// TIA Portal V19 export
FUNCTION "INTERLOCK" : Void   // FC7, LAD
{ S7_Optimized_Access := 'TRUE' }
// stored: SetENOAutomatically false
   VAR_TEMP   // added for the SCL form of the ladder/FBD networks
      _w1 : Bool;
      _w2 : Bool;
   END_VAR
BEGIN

REGION Network 1: ERROR
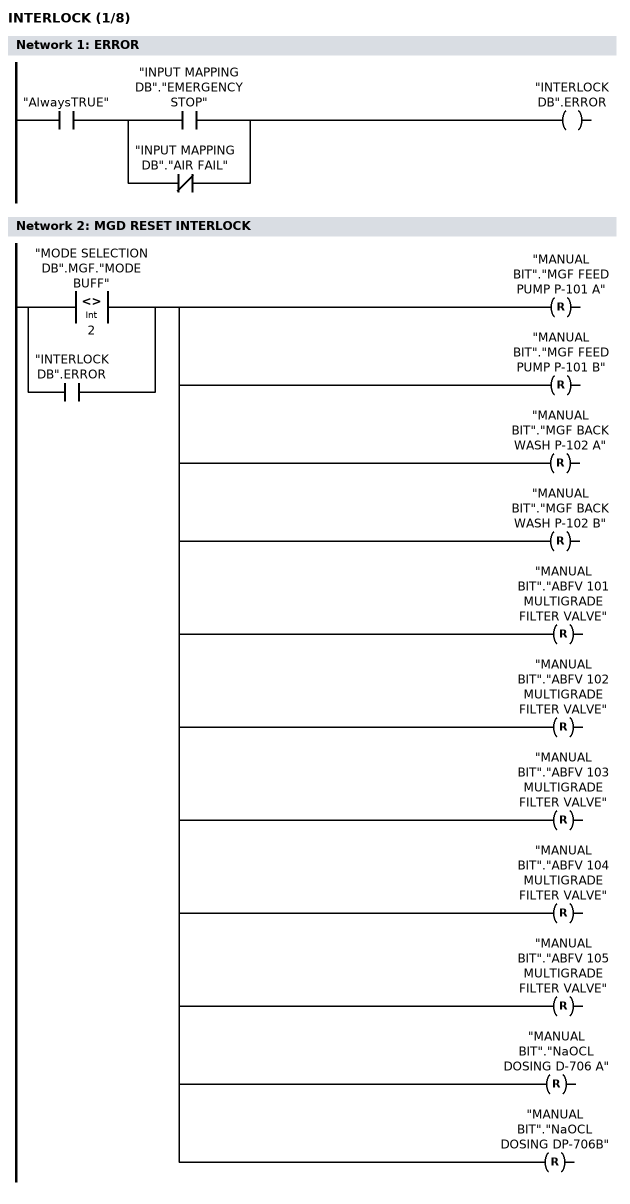
   RUNG wire#powerrail
      Contact( "AlwaysTRUE" )
      wire#w1
      Contact( "INPUT MAPPING DB"."EMERGENCY STOP" )
      wire#w2
      Coil( "INTERLOCK DB".ERROR )
   END_RUNG
   RUNG wire#w1
      I_Contact( "INPUT MAPPING DB"."AIR FAIL" )
   END_RUNG wire#w2
   // the same network as SCL:
   "INTERLOCK DB".ERROR := "AlwaysTRUE" AND ("INPUT MAPPING DB"."EMERGENCY STOP" OR NOT "INPUT MAPPING DB"."AIR FAIL");
END_REGION

REGION Network 2: MGD RESET INTERLOCK
   RUNG wire#powerrail
      { S7_Templates := "SrcType := Int" } NE_Contact(in1 := "MODE SELECTION DB".MGF."MODE BUFF", in2 := 2)
      wire#w1
      R_Coil( "MANUAL BIT"."MGF FEED PUMP P-101 A" )
   END_RUNG
   RUNG wire#powerrail
      Contact( "INTERLOCK DB".ERROR )
   END_RUNG wire#w1
   RUNG wire#w1
      R_Coil( "MANUAL BIT"."MGF FEED PUMP P-101 B" )
   END_RUNG
   RUNG wire#w1
      R_Coil( "MANUAL BIT"."MGF BACK WASH P-102 A" )
   END_RUNG
   RUNG wire#w1
      R_Coil( "MANUAL BIT"."MGF BACK WASH P-102 B" )
   END_RUNG
   RUNG wire#w1
      R_Coil( "MANUAL BIT"."ABFV 101 MULTIGRADE FILTER VALVE" )
   END_RUNG
   RUNG wire#w1
      R_Coil( "MANUAL BIT"."ABFV 102 MULTIGRADE FILTER VALVE" )
   END_RUNG
   RUNG wire#w1
      R_Coil( "MANUAL BIT"."ABFV 103 MULTIGRADE FILTER VALVE" )
   END_RUNG
   RUNG wire#w1
      R_Coil( "MANUAL BIT"."ABFV 104 MULTIGRADE FILTER VALVE" )
   END_RUNG
   RUNG wire#w1
      R_Coil( "MANUAL BIT"."ABFV 105 MULTIGRADE FILTER VALVE" )
   END_RUNG
   RUNG wire#w1
      R_Coil( "MANUAL BIT"."NaOCL DOSING D-706 A" )
   END_RUNG
   RUNG wire#w1
      R_Coil( "MANUAL BIT"."NaOCL DOSING DP-706B" )
   END_RUNG
   // the same network as SCL:
   IF ("MODE SELECTION DB".MGF."MODE BUFF" <> 2) OR "INTERLOCK DB".ERROR THEN
       "MANUAL BIT"."MGF FEED PUMP P-101 A" := FALSE;
       "MANUAL BIT"."MGF FEED PUMP P-101 B" := FALSE;
       "MANUAL BIT"."MGF BACK WASH P-102 A" := FALSE;
       "MANUAL BIT"."MGF BACK WASH P-102 B" := FALSE;
       "MANUAL BIT"."ABFV 101 MULTIGRADE FILTER VALVE" := FALSE;
       "MANUAL BIT"."ABFV 102 MULTIGRADE FILTER VALVE" := FALSE;
       "MANUAL BIT"."ABFV 103 MULTIGRADE FILTER VALVE" := FALSE;
       "MANUAL BIT"."ABFV 104 MULTIGRADE FILTER VALVE" := FALSE;
       "MANUAL BIT"."ABFV 105 MULTIGRADE FILTER VALVE" := FALSE;
       "MANUAL BIT"."NaOCL DOSING D-706 A" := FALSE;
       "MANUAL BIT"."NaOCL DOSING DP-706B" := FALSE;
   END_IF;
END_REGION

REGION Network 3: UF RESET INTERLOCK
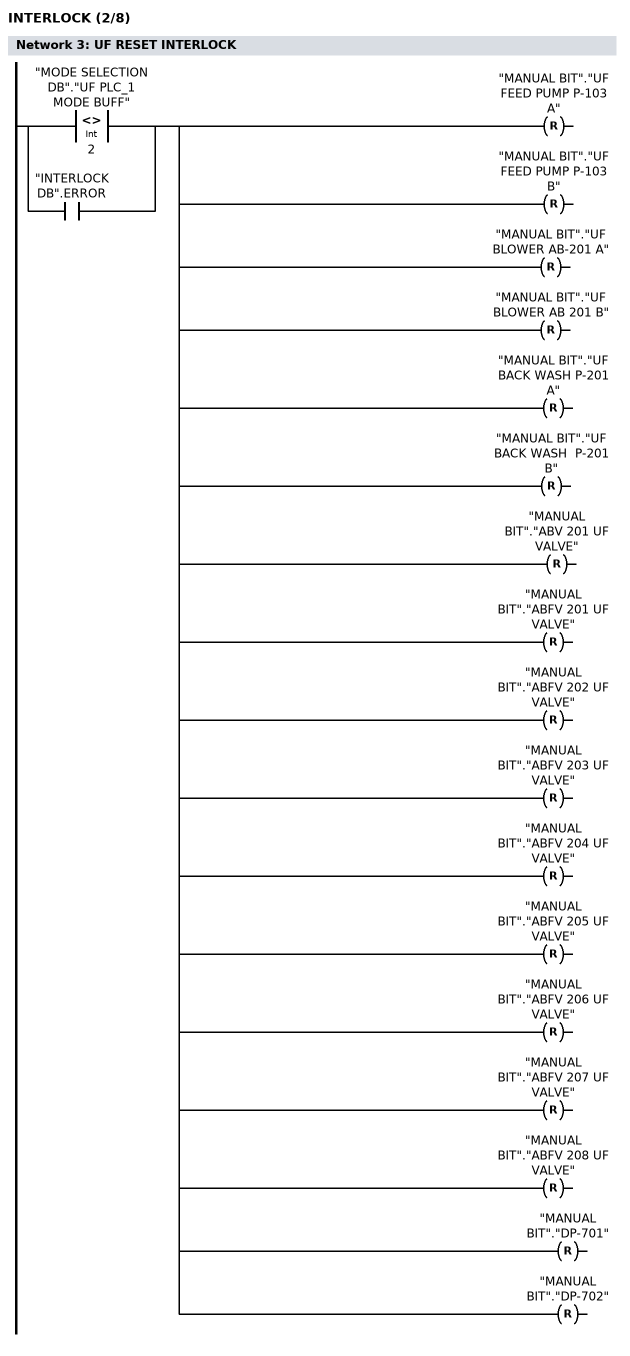
   RUNG wire#powerrail
      { S7_Templates := "SrcType := Int" } NE_Contact(in1 := "MODE SELECTION DB"."UF PLC_1 MODE BUFF", in2 := 2)
      wire#w1
      R_Coil( "MANUAL BIT"."UF FEED PUMP P-103 A" )
   END_RUNG
   RUNG wire#powerrail
      Contact( "INTERLOCK DB".ERROR )
   END_RUNG wire#w1
   RUNG wire#w1
      R_Coil( "MANUAL BIT"."UF FEED PUMP P-103 B" )
   END_RUNG
   RUNG wire#w1
      R_Coil( "MANUAL BIT"."UF BLOWER AB-201 A" )
   END_RUNG
   RUNG wire#w1
      R_Coil( "MANUAL BIT"."UF BLOWER AB 201 B" )
   END_RUNG
   RUNG wire#w1
      R_Coil( "MANUAL BIT"."UF BACK WASH P-201 A" )
   END_RUNG
   RUNG wire#w1
      R_Coil( "MANUAL BIT"."UF BACK WASH  P-201 B" )
   END_RUNG
   RUNG wire#w1
      R_Coil( "MANUAL BIT"."ABV 201 UF VALVE" )
   END_RUNG
   RUNG wire#w1
      R_Coil( "MANUAL BIT"."ABFV 201 UF VALVE" )
   END_RUNG
   RUNG wire#w1
      R_Coil( "MANUAL BIT"."ABFV 202 UF VALVE" )
   END_RUNG
   RUNG wire#w1
      R_Coil( "MANUAL BIT"."ABFV 203 UF VALVE" )
   END_RUNG
   RUNG wire#w1
      R_Coil( "MANUAL BIT"."ABFV 204 UF VALVE" )
   END_RUNG
   RUNG wire#w1
      R_Coil( "MANUAL BIT"."ABFV 205 UF VALVE" )
   END_RUNG
   RUNG wire#w1
      R_Coil( "MANUAL BIT"."ABFV 206 UF VALVE" )
   END_RUNG
   RUNG wire#w1
      R_Coil( "MANUAL BIT"."ABFV 207 UF VALVE" )
   END_RUNG
   RUNG wire#w1
      R_Coil( "MANUAL BIT"."ABFV 208 UF VALVE" )
   END_RUNG
   RUNG wire#w1
      R_Coil( "MANUAL BIT"."DP-701" )
   END_RUNG
   RUNG wire#w1
      R_Coil( "MANUAL BIT"."DP-702" )
   END_RUNG
   // the same network as SCL:
   IF ("MODE SELECTION DB"."UF PLC_1 MODE BUFF" <> 2) OR "INTERLOCK DB".ERROR THEN
       "MANUAL BIT"."UF FEED PUMP P-103 A" := FALSE;
       "MANUAL BIT"."UF FEED PUMP P-103 B" := FALSE;
       "MANUAL BIT"."UF BLOWER AB-201 A" := FALSE;
       "MANUAL BIT"."UF BLOWER AB 201 B" := FALSE;
       "MANUAL BIT"."UF BACK WASH P-201 A" := FALSE;
       "MANUAL BIT"."UF BACK WASH  P-201 B" := FALSE;
       "MANUAL BIT"."ABV 201 UF VALVE" := FALSE;
       "MANUAL BIT"."ABFV 201 UF VALVE" := FALSE;
       "MANUAL BIT"."ABFV 202 UF VALVE" := FALSE;
       "MANUAL BIT"."ABFV 203 UF VALVE" := FALSE;
       "MANUAL BIT"."ABFV 204 UF VALVE" := FALSE;
       "MANUAL BIT"."ABFV 205 UF VALVE" := FALSE;
       "MANUAL BIT"."ABFV 206 UF VALVE" := FALSE;
       "MANUAL BIT"."ABFV 207 UF VALVE" := FALSE;
       "MANUAL BIT"."ABFV 208 UF VALVE" := FALSE;
       "MANUAL BIT"."DP-701" := FALSE;
       "MANUAL BIT"."DP-702" := FALSE;
   END_IF;
END_REGION

REGION Network 4: DM RESET INTERLOCK
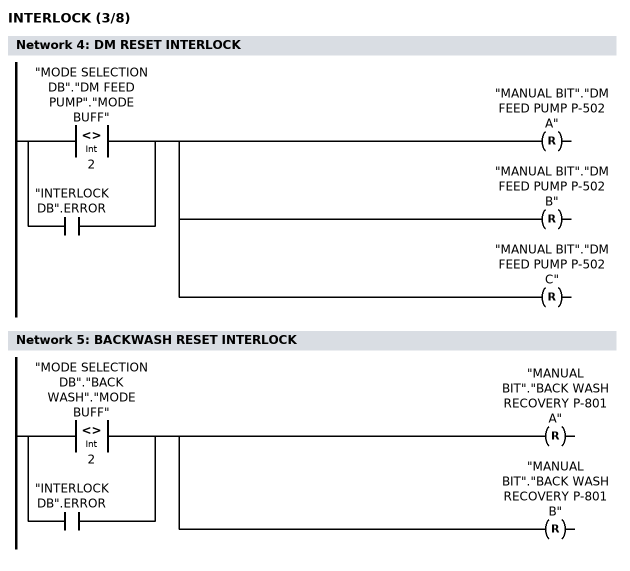
   RUNG wire#powerrail
      { S7_Templates := "SrcType := Int" } NE_Contact(in1 := "MODE SELECTION DB"."DM FEED PUMP"."MODE BUFF", in2 := 2)
      wire#w1
      R_Coil( "MANUAL BIT"."DM FEED PUMP P-502 A" )
   END_RUNG
   RUNG wire#powerrail
      Contact( "INTERLOCK DB".ERROR )
   END_RUNG wire#w1
   RUNG wire#w1
      R_Coil( "MANUAL BIT"."DM FEED PUMP P-502 B" )
   END_RUNG
   RUNG wire#w1
      R_Coil( "MANUAL BIT"."DM FEED PUMP P-502 C" )
   END_RUNG
   // the same network as SCL:
   IF ("MODE SELECTION DB"."DM FEED PUMP"."MODE BUFF" <> 2) OR "INTERLOCK DB".ERROR THEN
       "MANUAL BIT"."DM FEED PUMP P-502 A" := FALSE;
       "MANUAL BIT"."DM FEED PUMP P-502 B" := FALSE;
       "MANUAL BIT"."DM FEED PUMP P-502 C" := FALSE;
   END_IF;
END_REGION

REGION Network 5: BACKWASH RESET INTERLOCK
   RUNG wire#powerrail
      { S7_Templates := "SrcType := Int" } NE_Contact(in1 := "MODE SELECTION DB"."BACK WASH"."MODE BUFF", in2 := 2)
      wire#w1
      R_Coil( "MANUAL BIT"."BACK WASH RECOVERY P-801 A" )
   END_RUNG
   RUNG wire#powerrail
      Contact( "INTERLOCK DB".ERROR )
   END_RUNG wire#w1
   RUNG wire#w1
      R_Coil( "MANUAL BIT"."BACK WASH RECOVERY P-801 B" )
   END_RUNG
   // the same network as SCL:
   IF ("MODE SELECTION DB"."BACK WASH"."MODE BUFF" <> 2) OR "INTERLOCK DB".ERROR THEN
       "MANUAL BIT"."BACK WASH RECOVERY P-801 A" := FALSE;
       "MANUAL BIT"."BACK WASH RECOVERY P-801 B" := FALSE;
   END_IF;
END_REGION

REGION Network 6: SELECTION PUMP INTERLOCK_
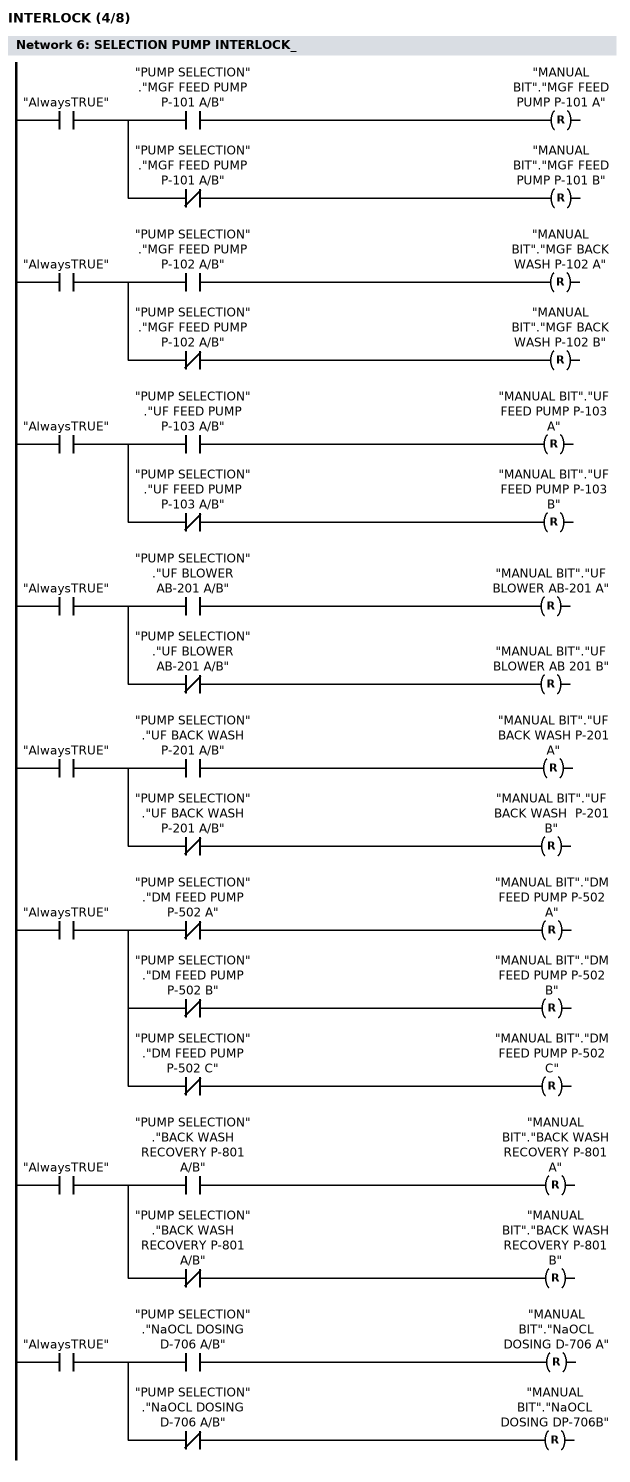
   RUNG wire#powerrail
      Contact( "AlwaysTRUE" )
      wire#w1
      Contact( "PUMP SELECTION"."MGF FEED PUMP P-101 A/B" )
      R_Coil( "MANUAL BIT"."MGF FEED PUMP P-101 A" )
   END_RUNG
   RUNG wire#w1
      I_Contact( "PUMP SELECTION"."MGF FEED PUMP P-101 A/B" )
      R_Coil( "MANUAL BIT"."MGF FEED PUMP P-101 B" )
   END_RUNG
   RUNG wire#powerrail
      Contact( "AlwaysTRUE" )
      wire#w2
      Contact( "PUMP SELECTION"."MGF FEED PUMP P-102 A/B" )
      R_Coil( "MANUAL BIT"."MGF BACK WASH P-102 A" )
   END_RUNG
   RUNG wire#w2
      I_Contact( "PUMP SELECTION"."MGF FEED PUMP P-102 A/B" )
      R_Coil( "MANUAL BIT"."MGF BACK WASH P-102 B" )
   END_RUNG
   RUNG wire#powerrail
      Contact( "AlwaysTRUE" )
      wire#w3
      Contact( "PUMP SELECTION"."UF FEED PUMP P-103 A/B" )
      R_Coil( "MANUAL BIT"."UF FEED PUMP P-103 A" )
   END_RUNG
   RUNG wire#w3
      I_Contact( "PUMP SELECTION"."UF FEED PUMP P-103 A/B" )
      R_Coil( "MANUAL BIT"."UF FEED PUMP P-103 B" )
   END_RUNG
   RUNG wire#powerrail
      Contact( "AlwaysTRUE" )
      wire#w4
      Contact( "PUMP SELECTION"."UF BLOWER AB-201 A/B" )
      R_Coil( "MANUAL BIT"."UF BLOWER AB-201 A" )
   END_RUNG
   RUNG wire#w4
      I_Contact( "PUMP SELECTION"."UF BLOWER AB-201 A/B" )
      R_Coil( "MANUAL BIT"."UF BLOWER AB 201 B" )
   END_RUNG
   RUNG wire#powerrail
      Contact( "AlwaysTRUE" )
      wire#w5
      Contact( "PUMP SELECTION"."UF BACK WASH P-201 A/B" )
      R_Coil( "MANUAL BIT"."UF BACK WASH P-201 A" )
   END_RUNG
   RUNG wire#w5
      I_Contact( "PUMP SELECTION"."UF BACK WASH P-201 A/B" )
      R_Coil( "MANUAL BIT"."UF BACK WASH  P-201 B" )
   END_RUNG
   RUNG wire#powerrail
      Contact( "AlwaysTRUE" )
      wire#w6
      I_Contact( "PUMP SELECTION"."DM FEED PUMP P-502 A" )
      R_Coil( "MANUAL BIT"."DM FEED PUMP P-502 A" )
   END_RUNG
   RUNG wire#w6
      I_Contact( "PUMP SELECTION"."DM FEED PUMP P-502 B" )
      R_Coil( "MANUAL BIT"."DM FEED PUMP P-502 B" )
   END_RUNG
   RUNG wire#w6
      I_Contact( "PUMP SELECTION"."DM FEED PUMP P-502 C" )
      R_Coil( "MANUAL BIT"."DM FEED PUMP P-502 C" )
   END_RUNG
   RUNG wire#powerrail
      Contact( "AlwaysTRUE" )
      wire#w7
      Contact( "PUMP SELECTION"."BACK WASH RECOVERY P-801 A/B" )
      R_Coil( "MANUAL BIT"."BACK WASH RECOVERY P-801 A" )
   END_RUNG
   RUNG wire#w7
      I_Contact( "PUMP SELECTION"."BACK WASH RECOVERY P-801 A/B" )
      R_Coil( "MANUAL BIT"."BACK WASH RECOVERY P-801 B" )
   END_RUNG
   RUNG wire#powerrail
      Contact( "AlwaysTRUE" )
      wire#w8
      Contact( "PUMP SELECTION"."NaOCL DOSING D-706 A/B" )
      R_Coil( "MANUAL BIT"."NaOCL DOSING D-706 A" )
   END_RUNG
   RUNG wire#w8
      I_Contact( "PUMP SELECTION"."NaOCL DOSING D-706 A/B" )
      R_Coil( "MANUAL BIT"."NaOCL DOSING DP-706B" )
   END_RUNG
   // the same network as SCL:
   IF "AlwaysTRUE" AND "PUMP SELECTION"."MGF FEED PUMP P-101 A/B" THEN
       "MANUAL BIT"."MGF FEED PUMP P-101 A" := FALSE;
   END_IF;
   IF "AlwaysTRUE" AND NOT "PUMP SELECTION"."MGF FEED PUMP P-101 A/B" THEN
       "MANUAL BIT"."MGF FEED PUMP P-101 B" := FALSE;
   END_IF;
   IF "AlwaysTRUE" AND "PUMP SELECTION"."MGF FEED PUMP P-102 A/B" THEN
       "MANUAL BIT"."MGF BACK WASH P-102 A" := FALSE;
   END_IF;
   IF "AlwaysTRUE" AND NOT "PUMP SELECTION"."MGF FEED PUMP P-102 A/B" THEN
       "MANUAL BIT"."MGF BACK WASH P-102 B" := FALSE;
   END_IF;
   IF "AlwaysTRUE" AND "PUMP SELECTION"."UF FEED PUMP P-103 A/B" THEN
       "MANUAL BIT"."UF FEED PUMP P-103 A" := FALSE;
   END_IF;
   IF "AlwaysTRUE" AND NOT "PUMP SELECTION"."UF FEED PUMP P-103 A/B" THEN
       "MANUAL BIT"."UF FEED PUMP P-103 B" := FALSE;
   END_IF;
   IF "AlwaysTRUE" AND "PUMP SELECTION"."UF BLOWER AB-201 A/B" THEN
       "MANUAL BIT"."UF BLOWER AB-201 A" := FALSE;
   END_IF;
   IF "AlwaysTRUE" AND NOT "PUMP SELECTION"."UF BLOWER AB-201 A/B" THEN
       "MANUAL BIT"."UF BLOWER AB 201 B" := FALSE;
   END_IF;
   IF "AlwaysTRUE" AND "PUMP SELECTION"."UF BACK WASH P-201 A/B" THEN
       "MANUAL BIT"."UF BACK WASH P-201 A" := FALSE;
   END_IF;
   IF "AlwaysTRUE" AND NOT "PUMP SELECTION"."UF BACK WASH P-201 A/B" THEN
       "MANUAL BIT"."UF BACK WASH  P-201 B" := FALSE;
   END_IF;
   IF "AlwaysTRUE" AND NOT "PUMP SELECTION"."DM FEED PUMP P-502 A" THEN
       "MANUAL BIT"."DM FEED PUMP P-502 A" := FALSE;
   END_IF;
   IF "AlwaysTRUE" AND NOT "PUMP SELECTION"."DM FEED PUMP P-502 B" THEN
       "MANUAL BIT"."DM FEED PUMP P-502 B" := FALSE;
   END_IF;
   IF "AlwaysTRUE" AND NOT "PUMP SELECTION"."DM FEED PUMP P-502 C" THEN
       "MANUAL BIT"."DM FEED PUMP P-502 C" := FALSE;
   END_IF;
   IF "AlwaysTRUE" AND "PUMP SELECTION"."BACK WASH RECOVERY P-801 A/B" THEN
       "MANUAL BIT"."BACK WASH RECOVERY P-801 A" := FALSE;
   END_IF;
   IF "AlwaysTRUE" AND NOT "PUMP SELECTION"."BACK WASH RECOVERY P-801 A/B" THEN
       "MANUAL BIT"."BACK WASH RECOVERY P-801 B" := FALSE;
   END_IF;
   IF "AlwaysTRUE" AND "PUMP SELECTION"."NaOCL DOSING D-706 A/B" THEN
       "MANUAL BIT"."NaOCL DOSING D-706 A" := FALSE;
   END_IF;
   IF "AlwaysTRUE" AND NOT "PUMP SELECTION"."NaOCL DOSING D-706 A/B" THEN
       "MANUAL BIT"."NaOCL DOSING DP-706B" := FALSE;
   END_IF;
END_REGION

REGION Network 9: AUTO__________________MGF PROCESS
END_REGION

REGION Network 10: PS-101.....................TAGE NHI MILA
END_REGION

REGION Network 11: PS201...........................
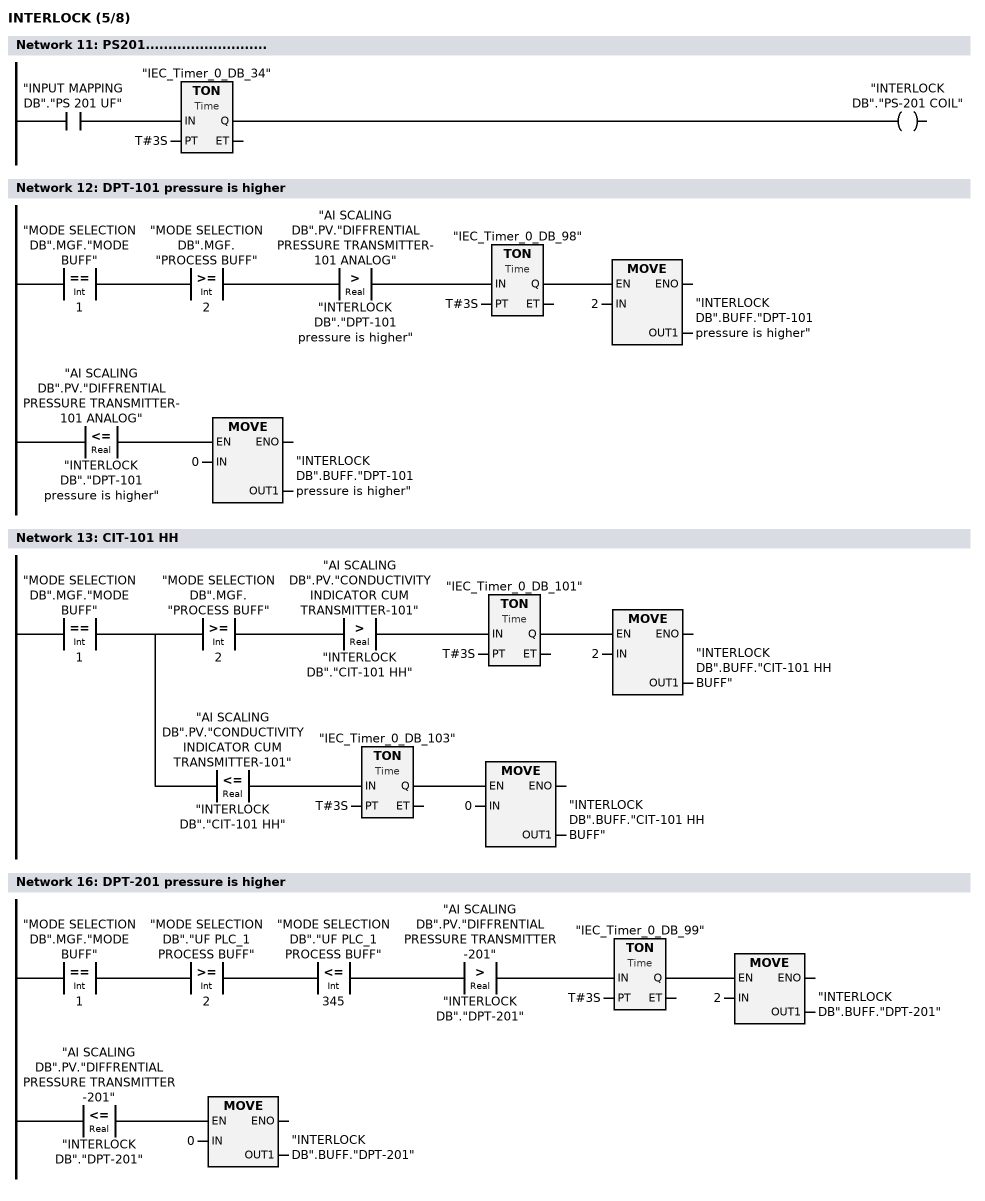
   RUNG wire#powerrail
      Contact( "INPUT MAPPING DB"."PS 201 UF" )
      { S7_Templates := "time_type := Time" } "IEC_Timer_0_DB_34".TON(pt := T#3S, et =>)
      Coil( "INTERLOCK DB"."PS-201 COIL" )
   END_RUNG
   // the same network as SCL:
   "IEC_Timer_0_DB_34".TON(IN := "INPUT MAPPING DB"."PS 201 UF", PT := T#3S);
   "INTERLOCK DB"."PS-201 COIL" := "IEC_Timer_0_DB_34".Q;
END_REGION

REGION Network 12: DPT-101 pressure is higher
   RUNG wire#powerrail
      { S7_Templates := "SrcType := Int" } EQ_Contact(in1 := "MODE SELECTION DB".MGF."MODE BUFF", in2 := 1)
      { S7_Templates := "SrcType := Int" } GE_Contact(in1 := "MODE SELECTION DB".MGF."PROCESS BUFF", in2 := 2)
      { S7_Templates := "SrcType := Real" } GT_Contact(in1 := "AI SCALING DB".PV."DIFFRENTIAL PRESSURE TRANSMITTER-101 ANALOG", in2 := "INTERLOCK DB"."DPT-101 pressure is higher")
      { S7_Templates := "time_type := Time" } "IEC_Timer_0_DB_98".TON(pt := T#3S, et =>)
      Move(in := 2, out1 => "INTERLOCK DB".BUFF."DPT-101 pressure is higher")
   END_RUNG
   RUNG wire#powerrail
      { S7_Templates := "SrcType := Real" } LE_Contact(in1 := "AI SCALING DB".PV."DIFFRENTIAL PRESSURE TRANSMITTER-101 ANALOG", in2 := "INTERLOCK DB"."DPT-101 pressure is higher")
      Move(in := 0, out1 => "INTERLOCK DB".BUFF."DPT-101 pressure is higher")
   END_RUNG
   // the same network as SCL:
   "IEC_Timer_0_DB_98".TON(IN := ("MODE SELECTION DB".MGF."MODE BUFF" = 1) AND ("MODE SELECTION DB".MGF."PROCESS BUFF" >= 2) AND ("AI SCALING DB".PV."DIFFRENTIAL PRESSURE TRANSMITTER-101 ANALOG" > "INTERLOCK DB"."DPT-101 pressure is higher"),
                           PT := T#3S);
   IF "IEC_Timer_0_DB_98".Q THEN "INTERLOCK DB".BUFF."DPT-101 pressure is higher" := 2; END_IF;
   IF "AI SCALING DB".PV."DIFFRENTIAL PRESSURE TRANSMITTER-101 ANALOG" <= "INTERLOCK DB"."DPT-101 pressure is higher" THEN
       "INTERLOCK DB".BUFF."DPT-101 pressure is higher" := 0;
   END_IF;
END_REGION

REGION Network 13: CIT-101 HH
   RUNG wire#powerrail
      { S7_Templates := "SrcType := Int" } EQ_Contact(in1 := "MODE SELECTION DB".MGF."MODE BUFF", in2 := 1)
      wire#w1
      { S7_Templates := "SrcType := Int" } GE_Contact(in1 := "MODE SELECTION DB".MGF."PROCESS BUFF", in2 := 2)
      { S7_Templates := "SrcType := Real" } GT_Contact(in1 := "AI SCALING DB".PV."CONDUCTIVITY INDICATOR CUM TRANSMITTER-101", in2 := "INTERLOCK DB"."CIT-101 HH")
      { S7_Templates := "time_type := Time" } "IEC_Timer_0_DB_101".TON(pt := T#3S, et =>)
      Move(in := 2, out1 => "INTERLOCK DB".BUFF."CIT-101 HH BUFF")
   END_RUNG
   RUNG wire#w1
      { S7_Templates := "SrcType := Real" } LE_Contact(in1 := "AI SCALING DB".PV."CONDUCTIVITY INDICATOR CUM TRANSMITTER-101", in2 := "INTERLOCK DB"."CIT-101 HH")
      { S7_Templates := "time_type := Time" } "IEC_Timer_0_DB_103".TON(pt := T#3S, et =>)
      Move(in := 0, out1 => "INTERLOCK DB".BUFF."CIT-101 HH BUFF")
   END_RUNG
   // the same network as SCL:
   #_w1 := "MODE SELECTION DB".MGF."MODE BUFF" = 1;
   "IEC_Timer_0_DB_101".TON(IN := #_w1 AND ("MODE SELECTION DB".MGF."PROCESS BUFF" >= 2) AND ("AI SCALING DB".PV."CONDUCTIVITY INDICATOR CUM TRANSMITTER-101" > "INTERLOCK DB"."CIT-101 HH"),
                           PT := T#3S);
   IF "IEC_Timer_0_DB_101".Q THEN "INTERLOCK DB".BUFF."CIT-101 HH BUFF" := 2; END_IF;
   "IEC_Timer_0_DB_103".TON(IN := #_w1 AND ("AI SCALING DB".PV."CONDUCTIVITY INDICATOR CUM TRANSMITTER-101" <= "INTERLOCK DB"."CIT-101 HH"),
                           PT := T#3S);
   IF "IEC_Timer_0_DB_103".Q THEN "INTERLOCK DB".BUFF."CIT-101 HH BUFF" := 0; END_IF;
END_REGION

REGION Network 15: AUTO__________________UF PROCESS
END_REGION

REGION Network 16: DPT-201 pressure is higher
   RUNG wire#powerrail
      { S7_Templates := "SrcType := Int" } EQ_Contact(in1 := "MODE SELECTION DB".MGF."MODE BUFF", in2 := 1)
      { S7_Templates := "SrcType := Int" } GE_Contact(in1 := "MODE SELECTION DB"."UF PLC_1 PROCESS BUFF", in2 := 2)
      { S7_Templates := "SrcType := Int" } LE_Contact(in1 := "MODE SELECTION DB"."UF PLC_1 PROCESS BUFF", in2 := 345)
      { S7_Templates := "SrcType := Real" } GT_Contact(in1 := "AI SCALING DB".PV."DIFFRENTIAL PRESSURE TRANSMITTER-201", in2 := "INTERLOCK DB"."DPT-201")
      { S7_Templates := "time_type := Time" } "IEC_Timer_0_DB_99".TON(pt := T#3S, et =>)
      Move(in := 2, out1 => "INTERLOCK DB".BUFF."DPT-201")
   END_RUNG
   RUNG wire#powerrail
      { S7_Templates := "SrcType := Real" } LE_Contact(in1 := "AI SCALING DB".PV."DIFFRENTIAL PRESSURE TRANSMITTER-201", in2 := "INTERLOCK DB"."DPT-201")
      Move(in := 0, out1 => "INTERLOCK DB".BUFF."DPT-201")
   END_RUNG
   // the same network as SCL:
   "IEC_Timer_0_DB_99".TON(IN := ("MODE SELECTION DB".MGF."MODE BUFF" = 1) AND ("MODE SELECTION DB"."UF PLC_1 PROCESS BUFF" >= 2) AND ("MODE SELECTION DB"."UF PLC_1 PROCESS BUFF" <= 345) AND ("AI SCALING DB".PV."DIFFRENTIAL PRESSURE TRANSMITTER-201" > "INTERLOCK DB"."DPT-201"),
                           PT := T#3S);
   IF "IEC_Timer_0_DB_99".Q THEN "INTERLOCK DB".BUFF."DPT-201" := 2; END_IF;
   IF "AI SCALING DB".PV."DIFFRENTIAL PRESSURE TRANSMITTER-201" <= "INTERLOCK DB"."DPT-201" THEN
       "INTERLOCK DB".BUFF."DPT-201" := 0;
   END_IF;
END_REGION

REGION Network 17: UF INTERLOCK FOR LT-102 AND LT201 SYSTER PAUSE
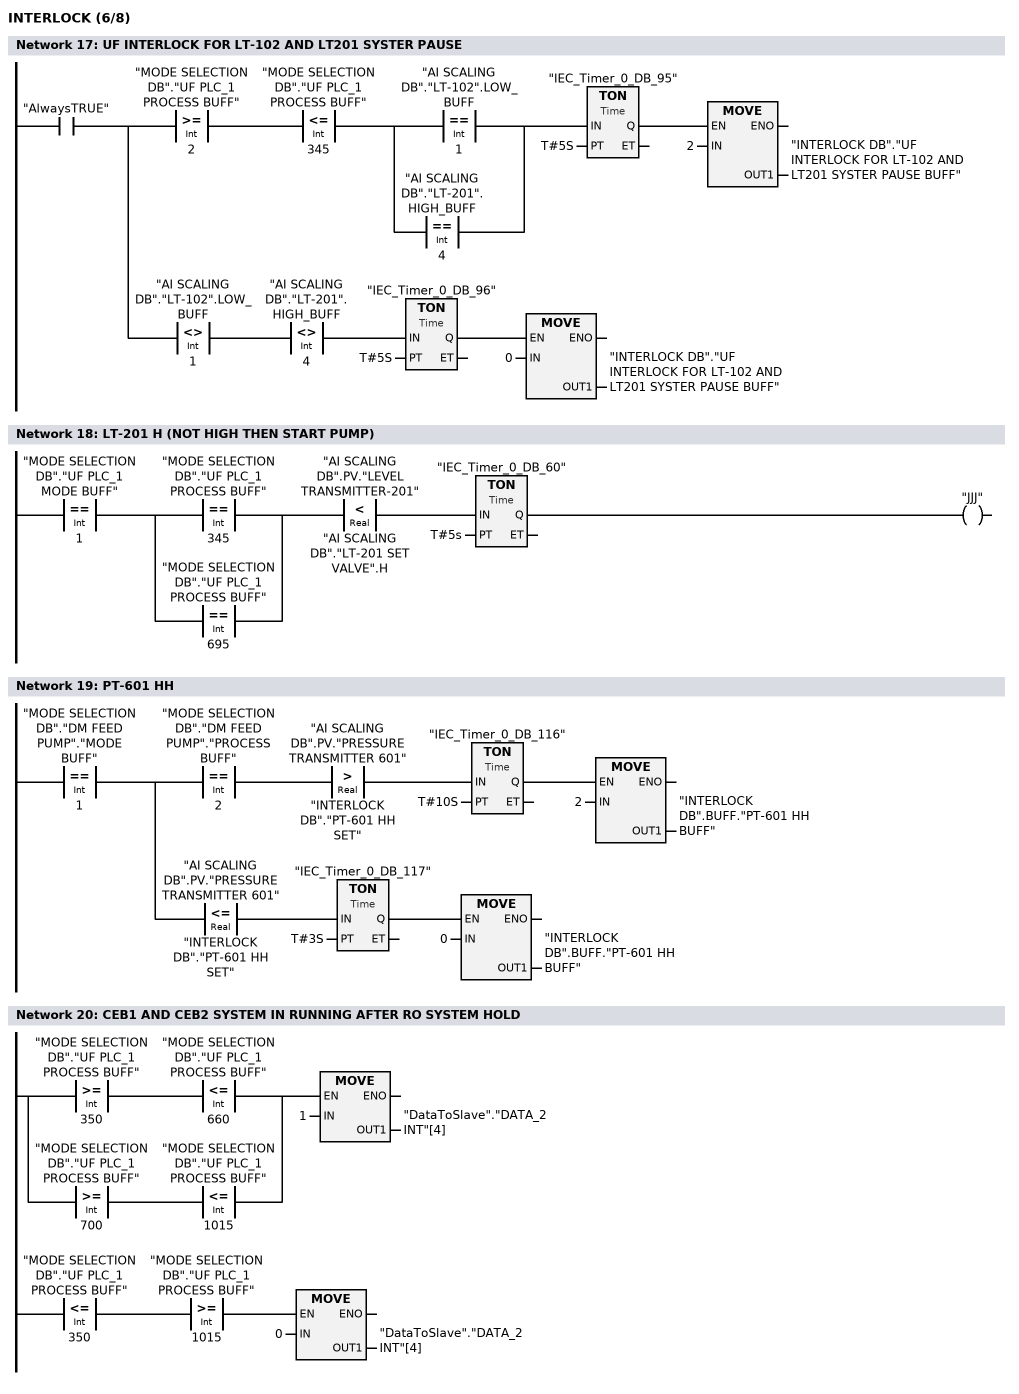
   RUNG wire#powerrail
      Contact( "AlwaysTRUE" )
      wire#w1
      { S7_Templates := "SrcType := Int" } GE_Contact(in1 := "MODE SELECTION DB"."UF PLC_1 PROCESS BUFF", in2 := 2)
      { S7_Templates := "SrcType := Int" } LE_Contact(in1 := "MODE SELECTION DB"."UF PLC_1 PROCESS BUFF", in2 := 345)
      wire#w2
      { S7_Templates := "SrcType := Int" } EQ_Contact(in1 := "AI SCALING DB"."LT-102".LOW_BUFF, in2 := 1)
      wire#w3
      { S7_Templates := "time_type := Time" } "IEC_Timer_0_DB_95".TON(pt := T#5S, et =>)
      Move(in := 2, out1 => "INTERLOCK DB"."UF INTERLOCK FOR LT-102 AND LT201 SYSTER PAUSE BUFF")
   END_RUNG
   RUNG wire#w2
      { S7_Templates := "SrcType := Int" } EQ_Contact(in1 := "AI SCALING DB"."LT-201".HIGH_BUFF, in2 := 4)
   END_RUNG wire#w3
   RUNG wire#w1
      { S7_Templates := "SrcType := Int" } NE_Contact(in1 := "AI SCALING DB"."LT-102".LOW_BUFF, in2 := 1)
      { S7_Templates := "SrcType := Int" } NE_Contact(in1 := "AI SCALING DB"."LT-201".HIGH_BUFF, in2 := 4)
      { S7_Templates := "time_type := Time" } "IEC_Timer_0_DB_96".TON(pt := T#5S, et =>)
      Move(in := 0, out1 => "INTERLOCK DB"."UF INTERLOCK FOR LT-102 AND LT201 SYSTER PAUSE BUFF")
   END_RUNG
   // the same network as SCL:
   "IEC_Timer_0_DB_95".TON(IN := "AlwaysTRUE" AND ("MODE SELECTION DB"."UF PLC_1 PROCESS BUFF" >= 2) AND ("MODE SELECTION DB"."UF PLC_1 PROCESS BUFF" <= 345) AND (("AI SCALING DB"."LT-102".LOW_BUFF = 1) OR ("AI SCALING DB"."LT-201".HIGH_BUFF = 4)),
                           PT := T#5S);
   IF "IEC_Timer_0_DB_95".Q THEN
       "INTERLOCK DB"."UF INTERLOCK FOR LT-102 AND LT201 SYSTER PAUSE BUFF" := 2;
   END_IF;
   "IEC_Timer_0_DB_96".TON(IN := "AlwaysTRUE" AND ("AI SCALING DB"."LT-102".LOW_BUFF <> 1) AND ("AI SCALING DB"."LT-201".HIGH_BUFF <> 4),
                           PT := T#5S);
   IF "IEC_Timer_0_DB_96".Q THEN
       "INTERLOCK DB"."UF INTERLOCK FOR LT-102 AND LT201 SYSTER PAUSE BUFF" := 0;
   END_IF;
END_REGION

REGION Network 18: LT-201 H (NOT HIGH THEN START PUMP)
   RUNG wire#powerrail
      { S7_Templates := "SrcType := Int" } EQ_Contact(in1 := "MODE SELECTION DB"."UF PLC_1 MODE BUFF", in2 := 1)
      wire#w1
      { S7_Templates := "SrcType := Int" } EQ_Contact(in1 := "MODE SELECTION DB"."UF PLC_1 PROCESS BUFF", in2 := 345)
      wire#w2
      { S7_Templates := "SrcType := Real" } LT_Contact(in1 := "AI SCALING DB".PV."LEVEL TRANSMITTER-201", in2 := "AI SCALING DB"."LT-201 SET VALVE".H)
      { S7_Templates := "time_type := Time" } "IEC_Timer_0_DB_60".TON(pt := T#5s, et =>)
      Coil( "JJJ" )
   END_RUNG
   RUNG wire#w1
      { S7_Templates := "SrcType := Int" } EQ_Contact(in1 := "MODE SELECTION DB"."UF PLC_1 PROCESS BUFF", in2 := 695)
   END_RUNG wire#w2
   // the same network as SCL:
   "IEC_Timer_0_DB_60".TON(IN := ("MODE SELECTION DB"."UF PLC_1 MODE BUFF" = 1) AND (("MODE SELECTION DB"."UF PLC_1 PROCESS BUFF" = 345) OR ("MODE SELECTION DB"."UF PLC_1 PROCESS BUFF" = 695)) AND ("AI SCALING DB".PV."LEVEL TRANSMITTER-201" < "AI SCALING DB"."LT-201 SET VALVE".H),
                           PT := T#5s);
   "JJJ" := "IEC_Timer_0_DB_60".Q;
END_REGION

REGION Network 19: PT-601 HH
   RUNG wire#powerrail
      { S7_Templates := "SrcType := Int" } EQ_Contact(in1 := "MODE SELECTION DB"."DM FEED PUMP"."MODE BUFF", in2 := 1)
      wire#w1
      { S7_Templates := "SrcType := Int" } EQ_Contact(in1 := "MODE SELECTION DB"."DM FEED PUMP"."PROCESS BUFF", in2 := 2)
      { S7_Templates := "SrcType := Real" } GT_Contact(in1 := "AI SCALING DB".PV."PRESSURE TRANSMITTER 601", in2 := "INTERLOCK DB"."PT-601 HH SET")
      { S7_Templates := "time_type := Time" } "IEC_Timer_0_DB_116".TON(pt := T#10S, et =>)
      Move(in := 2, out1 => "INTERLOCK DB".BUFF."PT-601 HH BUFF")
   END_RUNG
   RUNG wire#w1
      { S7_Templates := "SrcType := Real" } LE_Contact(in1 := "AI SCALING DB".PV."PRESSURE TRANSMITTER 601", in2 := "INTERLOCK DB"."PT-601 HH SET")
      { S7_Templates := "time_type := Time" } "IEC_Timer_0_DB_117".TON(pt := T#3S, et =>)
      Move(in := 0, out1 => "INTERLOCK DB".BUFF."PT-601 HH BUFF")
   END_RUNG
   // the same network as SCL:
   #_w1 := "MODE SELECTION DB"."DM FEED PUMP"."MODE BUFF" = 1;
   "IEC_Timer_0_DB_116".TON(IN := #_w1 AND ("MODE SELECTION DB"."DM FEED PUMP"."PROCESS BUFF" = 2) AND ("AI SCALING DB".PV."PRESSURE TRANSMITTER 601" > "INTERLOCK DB"."PT-601 HH SET"),
                           PT := T#10S);
   IF "IEC_Timer_0_DB_116".Q THEN "INTERLOCK DB".BUFF."PT-601 HH BUFF" := 2; END_IF;
   "IEC_Timer_0_DB_117".TON(IN := #_w1 AND ("AI SCALING DB".PV."PRESSURE TRANSMITTER 601" <= "INTERLOCK DB"."PT-601 HH SET"),
                           PT := T#3S);
   IF "IEC_Timer_0_DB_117".Q THEN "INTERLOCK DB".BUFF."PT-601 HH BUFF" := 0; END_IF;
END_REGION

REGION Network 20: CEB1 AND CEB2 SYSTEM IN RUNNING AFTER RO SYSTEM HOLD
   RUNG wire#powerrail
      { S7_Templates := "SrcType := Int" } GE_Contact(in1 := "MODE SELECTION DB"."UF PLC_1 PROCESS BUFF", in2 := 350)
      { S7_Templates := "SrcType := Int" } LE_Contact(in1 := "MODE SELECTION DB"."UF PLC_1 PROCESS BUFF", in2 := 660)
      wire#w1
      Move(in := 1, out1 => "DataToSlave"."DATA_2 INT"[4])
   END_RUNG
   RUNG wire#powerrail
      { S7_Templates := "SrcType := Int" } GE_Contact(in1 := "MODE SELECTION DB"."UF PLC_1 PROCESS BUFF", in2 := 700)
      { S7_Templates := "SrcType := Int" } LE_Contact(in1 := "MODE SELECTION DB"."UF PLC_1 PROCESS BUFF", in2 := 1015)
   END_RUNG wire#w1
   RUNG wire#powerrail
      { S7_Templates := "SrcType := Int" } LE_Contact(in1 := "MODE SELECTION DB"."UF PLC_1 PROCESS BUFF", in2 := 350)
      { S7_Templates := "SrcType := Int" } GE_Contact(in1 := "MODE SELECTION DB"."UF PLC_1 PROCESS BUFF", in2 := 1015)
      Move(in := 0, out1 => "DataToSlave"."DATA_2 INT"[4])
   END_RUNG
   // the same network as SCL:
   IF (("MODE SELECTION DB"."UF PLC_1 PROCESS BUFF" >= 350) AND ("MODE SELECTION DB"."UF PLC_1 PROCESS BUFF" <= 660)) OR (("MODE SELECTION DB"."UF PLC_1 PROCESS BUFF" >= 700) AND ("MODE SELECTION DB"."UF PLC_1 PROCESS BUFF" <= 1015)) THEN
       "DataToSlave"."DATA_2 INT"[4] := 1;
   END_IF;
   IF ("MODE SELECTION DB"."UF PLC_1 PROCESS BUFF" <= 350) AND ("MODE SELECTION DB"."UF PLC_1 PROCESS BUFF" >= 1015) THEN
       "DataToSlave"."DATA_2 INT"[4] := 0;
   END_IF;
END_REGION

REGION Network 22: AUTO__________________DM WATER TRANSFER
END_REGION

REGION Network 23: pHIT-601 LOW / HIGH
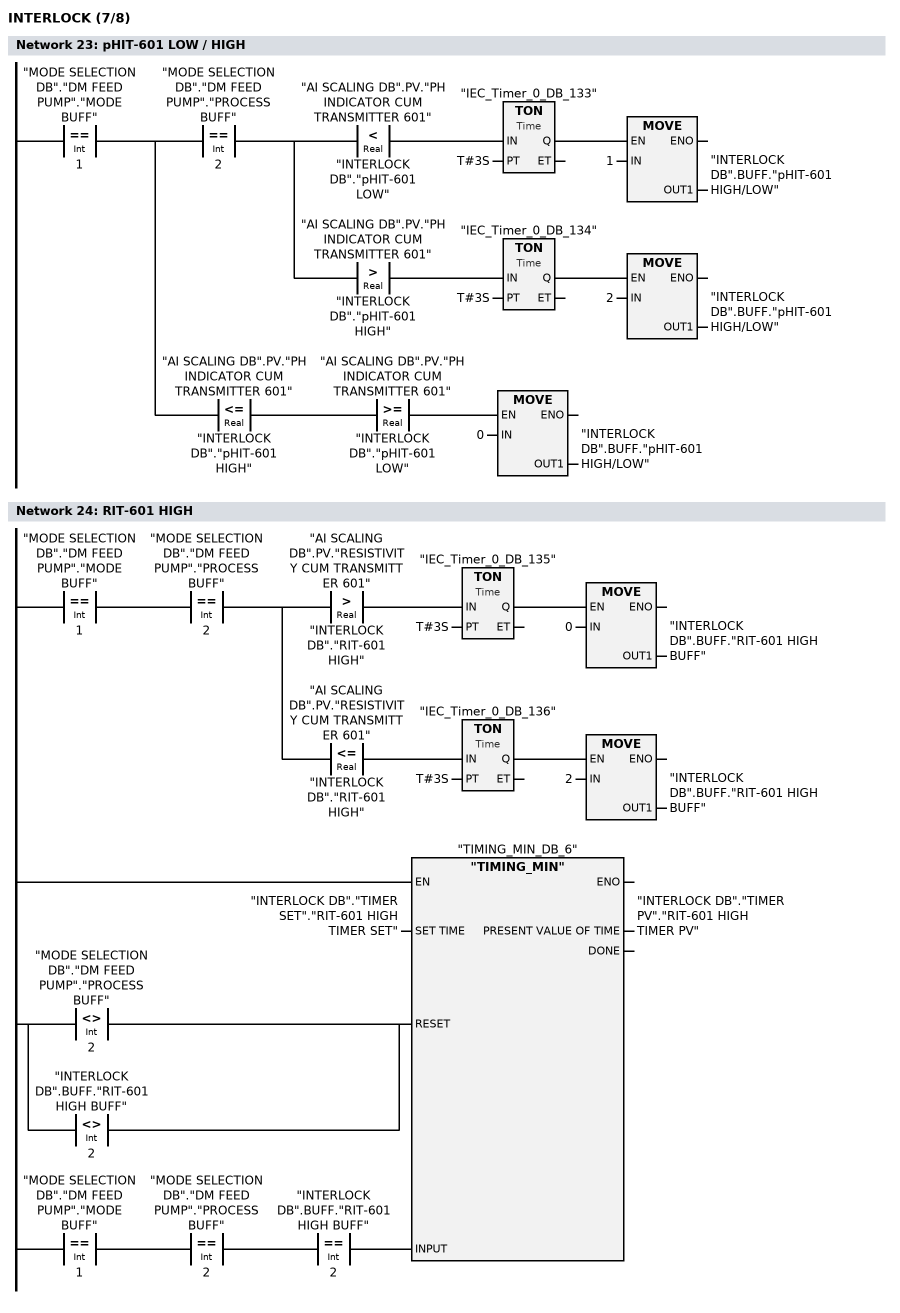
   RUNG wire#powerrail
      { S7_Templates := "SrcType := Int" } EQ_Contact(in1 := "MODE SELECTION DB"."DM FEED PUMP"."MODE BUFF", in2 := 1)
      wire#w1
      { S7_Templates := "SrcType := Int" } EQ_Contact(in1 := "MODE SELECTION DB"."DM FEED PUMP"."PROCESS BUFF", in2 := 2)
      wire#w2
      { S7_Templates := "SrcType := Real" } LT_Contact(in1 := "AI SCALING DB".PV."PH INDICATOR CUM TRANSMITTER 601", in2 := "INTERLOCK DB"."pHIT-601 LOW")
      { S7_Templates := "time_type := Time" } "IEC_Timer_0_DB_133".TON(pt := T#3S, et =>)
      Move(in := 1, out1 => "INTERLOCK DB".BUFF."pHIT-601 HIGH/LOW")
   END_RUNG
   RUNG wire#w2
      { S7_Templates := "SrcType := Real" } GT_Contact(in1 := "AI SCALING DB".PV."PH INDICATOR CUM TRANSMITTER 601", in2 := "INTERLOCK DB"."pHIT-601 HIGH")
      { S7_Templates := "time_type := Time" } "IEC_Timer_0_DB_134".TON(pt := T#3S, et =>)
      Move(in := 2, out1 => "INTERLOCK DB".BUFF."pHIT-601 HIGH/LOW")
   END_RUNG
   RUNG wire#w1
      { S7_Templates := "SrcType := Real" } LE_Contact(in1 := "AI SCALING DB".PV."PH INDICATOR CUM TRANSMITTER 601", in2 := "INTERLOCK DB"."pHIT-601 HIGH")
      { S7_Templates := "SrcType := Real" } GE_Contact(in1 := "AI SCALING DB".PV."PH INDICATOR CUM TRANSMITTER 601", in2 := "INTERLOCK DB"."pHIT-601 LOW")
      Move(in := 0, out1 => "INTERLOCK DB".BUFF."pHIT-601 HIGH/LOW")
   END_RUNG
   // the same network as SCL:
   #_w1 := "MODE SELECTION DB"."DM FEED PUMP"."MODE BUFF" = 1;
   #_w2 := #_w1 AND ("MODE SELECTION DB"."DM FEED PUMP"."PROCESS BUFF" = 2);
   "IEC_Timer_0_DB_133".TON(IN := #_w2 AND ("AI SCALING DB".PV."PH INDICATOR CUM TRANSMITTER 601" < "INTERLOCK DB"."pHIT-601 LOW"),
                           PT := T#3S);
   IF "IEC_Timer_0_DB_133".Q THEN "INTERLOCK DB".BUFF."pHIT-601 HIGH/LOW" := 1; END_IF;
   "IEC_Timer_0_DB_134".TON(IN := #_w2 AND ("AI SCALING DB".PV."PH INDICATOR CUM TRANSMITTER 601" > "INTERLOCK DB"."pHIT-601 HIGH"),
                           PT := T#3S);
   IF "IEC_Timer_0_DB_134".Q THEN "INTERLOCK DB".BUFF."pHIT-601 HIGH/LOW" := 2; END_IF;
   IF #_w1 AND ("AI SCALING DB".PV."PH INDICATOR CUM TRANSMITTER 601" <= "INTERLOCK DB"."pHIT-601 HIGH") AND ("AI SCALING DB".PV."PH INDICATOR CUM TRANSMITTER 601" >= "INTERLOCK DB"."pHIT-601 LOW") THEN
       "INTERLOCK DB".BUFF."pHIT-601 HIGH/LOW" := 0;
   END_IF;
END_REGION

REGION Network 24: RIT-601 HIGH
   RUNG wire#powerrail
      { S7_Templates := "SrcType := Int" } EQ_Contact(in1 := "MODE SELECTION DB"."DM FEED PUMP"."MODE BUFF", in2 := 1)
      { S7_Templates := "SrcType := Int" } EQ_Contact(in1 := "MODE SELECTION DB"."DM FEED PUMP"."PROCESS BUFF", in2 := 2)
      wire#w1
      { S7_Templates := "SrcType := Real" } GT_Contact(in1 := "AI SCALING DB".PV."RESISTIVITY CUM TRANSMITTER 601", in2 := "INTERLOCK DB"."RIT-601 HIGH")
      { S7_Templates := "time_type := Time" } "IEC_Timer_0_DB_135".TON(pt := T#3S, et =>)
      Move(in := 0, out1 => "INTERLOCK DB".BUFF."RIT-601 HIGH BUFF")
   END_RUNG
   RUNG wire#w1
      { S7_Templates := "SrcType := Real" } LE_Contact(in1 := "AI SCALING DB".PV."RESISTIVITY CUM TRANSMITTER 601", in2 := "INTERLOCK DB"."RIT-601 HIGH")
      { S7_Templates := "time_type := Time" } "IEC_Timer_0_DB_136".TON(pt := T#3S, et =>)
      Move(in := 2, out1 => "INTERLOCK DB".BUFF."RIT-601 HIGH BUFF")
   END_RUNG
   RUNG wire#powerrail
      "TIMING_MIN_DB_6"(RESET := wire#w2, INPUT := wire#w3, "SET TIME" := "INTERLOCK DB"."TIMER SET"."RIT-601 HIGH TIMER SET", "PRESENT VALUE OF TIME" => "INTERLOCK DB"."TIMER PV"."RIT-601 HIGH TIMER PV", DONE =>)
   END_RUNG
   RUNG wire#powerrail
      { S7_Templates := "SrcType := Int" } NE_Contact(in1 := "MODE SELECTION DB"."DM FEED PUMP"."PROCESS BUFF", in2 := 2)
   END_RUNG wire#w2
   RUNG wire#powerrail
      { S7_Templates := "SrcType := Int" } NE_Contact(in1 := "INTERLOCK DB".BUFF."RIT-601 HIGH BUFF", in2 := 2)
   END_RUNG wire#w2
   RUNG wire#powerrail
      { S7_Templates := "SrcType := Int" } EQ_Contact(in1 := "MODE SELECTION DB"."DM FEED PUMP"."MODE BUFF", in2 := 1)
      { S7_Templates := "SrcType := Int" } EQ_Contact(in1 := "MODE SELECTION DB"."DM FEED PUMP"."PROCESS BUFF", in2 := 2)
      { S7_Templates := "SrcType := Int" } EQ_Contact(in1 := "INTERLOCK DB".BUFF."RIT-601 HIGH BUFF", in2 := 2)
   END_RUNG wire#w3
   // the same network as SCL:
   #_w1 := ("MODE SELECTION DB"."DM FEED PUMP"."MODE BUFF" = 1) AND ("MODE SELECTION DB"."DM FEED PUMP"."PROCESS BUFF" = 2);
   "IEC_Timer_0_DB_135".TON(IN := #_w1 AND ("AI SCALING DB".PV."RESISTIVITY CUM TRANSMITTER 601" > "INTERLOCK DB"."RIT-601 HIGH"),
                           PT := T#3S);
   IF "IEC_Timer_0_DB_135".Q THEN "INTERLOCK DB".BUFF."RIT-601 HIGH BUFF" := 0; END_IF;
   "IEC_Timer_0_DB_136".TON(IN := #_w1 AND ("AI SCALING DB".PV."RESISTIVITY CUM TRANSMITTER 601" <= "INTERLOCK DB"."RIT-601 HIGH"),
                           PT := T#3S);
   IF "IEC_Timer_0_DB_136".Q THEN "INTERLOCK DB".BUFF."RIT-601 HIGH BUFF" := 2; END_IF;
   "TIMING_MIN_DB_6"("SET TIME" := "INTERLOCK DB"."TIMER SET"."RIT-601 HIGH TIMER SET",   // "TIMING_MIN"
                     RESET := ("MODE SELECTION DB"."DM FEED PUMP"."PROCESS BUFF" <> 2) OR ("INTERLOCK DB".BUFF."RIT-601 HIGH BUFF" <> 2),
                     INPUT := ("MODE SELECTION DB"."DM FEED PUMP"."MODE BUFF" = 1) AND ("MODE SELECTION DB"."DM FEED PUMP"."PROCESS BUFF" = 2) AND ("INTERLOCK DB".BUFF."RIT-601 HIGH BUFF" = 2),
                     "PRESENT VALUE OF TIME" => "INTERLOCK DB"."TIMER PV"."RIT-601 HIGH TIMER PV");
END_REGION

REGION Network 25: UV ONLY ALARM
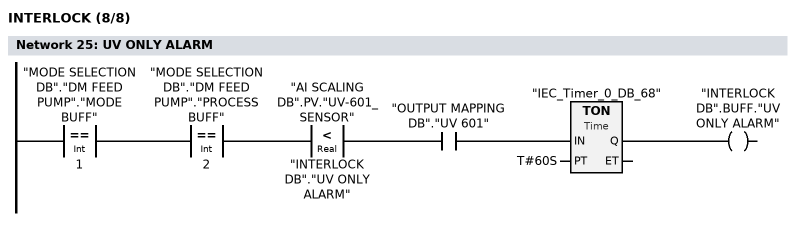
   RUNG wire#powerrail
      { S7_Templates := "SrcType := Int" } EQ_Contact(in1 := "MODE SELECTION DB"."DM FEED PUMP"."MODE BUFF", in2 := 1)
      { S7_Templates := "SrcType := Int" } EQ_Contact(in1 := "MODE SELECTION DB"."DM FEED PUMP"."PROCESS BUFF", in2 := 2)
      { S7_Templates := "SrcType := Real" } LT_Contact(in1 := "AI SCALING DB".PV."UV-601_SENSOR", in2 := "INTERLOCK DB"."UV ONLY ALARM")
      Contact( "OUTPUT MAPPING DB"."UV 601" )
      { S7_Templates := "time_type := Time" } "IEC_Timer_0_DB_68".TON(pt := T#60S, et =>)
      Coil( "INTERLOCK DB".BUFF."UV ONLY ALARM" )
   END_RUNG
   // the same network as SCL:
   "IEC_Timer_0_DB_68".TON(IN := ("MODE SELECTION DB"."DM FEED PUMP"."MODE BUFF" = 1) AND ("MODE SELECTION DB"."DM FEED PUMP"."PROCESS BUFF" = 2) AND ("AI SCALING DB".PV."UV-601_SENSOR" < "INTERLOCK DB"."UV ONLY ALARM") AND "OUTPUT MAPPING DB"."UV 601",
                           PT := T#60S);
   "INTERLOCK DB".BUFF."UV ONLY ALARM" := "IEC_Timer_0_DB_68".Q;
END_REGION
END_FUNCTION
